// TIA Portal V18 export
FUNCTION "DINTinSeconds_to_time" : Void   // FC9, FBD
{ S7_Optimized_Access := 'TRUE' }
VERSION : 0.1
// stored: AutoNumber true, IsIECCheckEnabled false, SetENOAutomatically false, UDAEnableTagReadback false
   VAR_INPUT
      in : DInt;
   END_VAR
   VAR_OUTPUT
      out : Time;
   END_VAR
   VAR_TEMP
      pt_dint_by_1000 : DInt;
   END_VAR
BEGIN

REGION Network 1
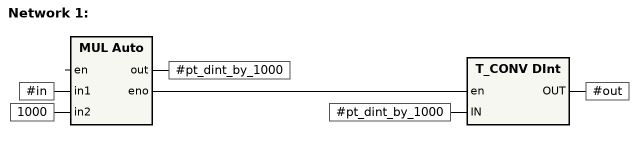
   #pt_dint_by_1000 := #in * 1000;
   T_CONV(IN := #pt_dint_by_1000, OUT => #out);
END_REGION
END_FUNCTION
